KUKA KRL data list: test_SCIRC.dat

&ACCESS RVP
&REL 2
&PARAM EDITMASK = *
&PARAM TEMPLATE = C:\KRC\Roboter\Template\vorgabe
&PARAM DISKPATH = KRC:\R1\Parcours\Nicolas F
DEFDAT test_SCIRC
;FOLD EXTERNAL DECLARATIONS;%{PE}%MKUKATPBASIS,%CEXT,%VCOMMON,%P
;FOLD BASISTECH EXT;%{PE}%MKUKATPBASIS,%CEXT,%VEXT,%P
EXT  BAS (BAS_COMMAND  :IN,REAL  :IN )
DECL INT SUCCESS
;ENDFOLD (BASISTECH EXT)
;FOLD USER EXT;%{E}%MKUKATPUSER,%CEXT,%VEXT,%P
;Make your modifications here

;ENDFOLD (USER EXT)
;ENDFOLD (EXTERNAL DECLARATIONS)

DECL E6POS XP1={X 838.869141,Y -277.480896, Z 609.890198,A 84.5815048,B -57.567028,C 91.0787354, S 2,T 10,E1 0.0,E2 0.0,E3 0.0,E4 0.0,E5 0.0,E6 0.0}
DECL E6POS XP2={X 1091.95776,Y -277.481,Z 851.570923, A 84.5815048,B -57.567028,C 91.0787354,S 2,T 10, E1 0.0,E2 0.0,E3 0.0,E4 0.0,E5 0.0,E6 0.0}
DECL FDAT FP2={TOOL_NO 4, BASE_NO 0,IPO_FRAME #BASE,POINT2[] " "}
DECL LDAT LCPDAT2= { VEL 2,ACC 100.000,APO_DIST 500.000,APO_FAC 50.0000,AXIS_VEL 100.000,AXIS_ACC 100.000,ORI_TYP #VAR,CIRC_TYP #BASE,JERK_FAC 50.0000,GEAR_JERK 100.000,EXAX_IGN 0,CB {AUX_PT {ORI #CONSIDER,E1 #CONSIDER,E2 #CONSIDER,E3 #CONSIDER,E4 #CONSIDER,E5 #CONSIDER,E6 #CONSIDER},TARGET_PT {ORI #INTERPOLATE,E1 #INTERPOLATE,E2 #INTERPOLATE,E3 #INTERPOLATE,E4 #INTERPOLATE,E5 #INTERPOLATE,E6 #INTERPOLATE} } }
DECL MODULEPARAM_T LAST_TP_PARAMS={PARAMS[] "Kuka.VelocityFieldEnabled=True;Kuka.ColDetectFieldEnabled=True;Kuka.MovementParameterFieldEnabled=True;Kuka.IsAngleEnabled=False;Kuka.PointName=P2;Kuka.FrameData.base_no=0;Kuka.FrameData.tool_no=4;Kuka.FrameData.ipo_frame=#BASE;Kuka.isglobalpoint=False;Kuka.MoveDataName=CPDAT1;Kuka.MovementData.cb={AUX_PT {ORI #CONSIDER,E1 #CONSIDER, E2 #CONSIDER,E3 #CONSIDER,E4 #CONSIDER,E5 #CONSIDER,E6 #CONSIDER}, TARGET_PT {ORI #INTERPOLATE,E1 #INTERPOLATE,E2 #INTERPOLATE, E3 #INTERPOLATE,E4 #INTERPOLATE,E5 #INTERPOLATE,E6 #INTERPOLATE} };Kuka.MovementData.apo_fac=50;Kuka.MovementData.apo_dist=500;Kuka.MovementData.axis_acc=100;Kuka.MovementData.axis_vel=100;Kuka.MovementData.circ_typ=#BASE;Kuka.MovementData.jerk_fac=50;Kuka.MovementData.ori_typ=#VAR;Kuka.MovementData.vel=2;Kuka.MovementData.acc=100;Kuka.MovementData.exax_ign=0;Kuka.VelocityPath=2;Kuka.BlendingEnabled=False;Kuka.APXEnabled=False;Kuka.CurrentCDSetIndex=0;Kuka.HelpPointName=P1"}
ENDDAT
